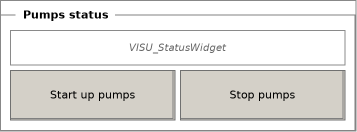
VISUALIZATION VISU_HydraulicsPumpsStatus  // 357x132
VAR_IN_OUT
	ref : Hydraulics;
    widget : HydraulicsWidget;
    ref_safety : SafetyHydraulics;
END_VAR
    Label (20,5 95x20), "Pumps status"
    Polyline (15,15) (0,15) (0,130) (355,130) (355,15) (115,15)
    Button (10,70 165x50), "Start up pumps", input disabled if: ref.processes.startUpPumps.statuses.enabledStatus.disabled
        OnMouseClick: execute { ref.processes.startUpPumps.do_request := TRUE; }
    Button (180,70 165x50), "Stop pumps", input disabled if: ref.processes.stopPumps.statuses.enabledStatus.disabled
        OnMouseClick: execute { ref.processes.stopPumps.do_request := TRUE; }
    Frame (10,30 335x35)
        shows VISU_StatusWidget(widget := widget.pumpsStatus)
END_VISUALIZATION

(* stored: Version 1.1.0.1, ProductVersion 3.1.4019.2
   Visu VISU_HydraulicsPumpsStatus: Id {bda26b11-bdb9-4025-b453-f0fb35eca0a3} *)
